RoboDK station: 直线500mm_v50.rdk

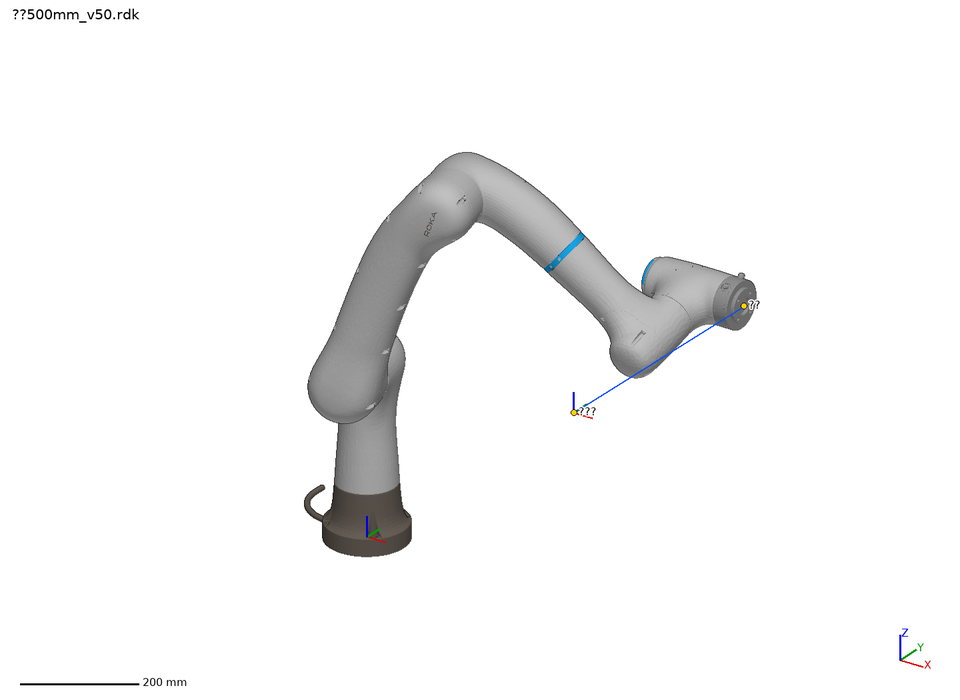
[picture v0: the station drawn from its stored meshes, robots at their saved joint values, targets as dots, program paths as lines]
Station 直线500mm_v50 (saved by RoboDK 5.9.0). Poses are relative to the parent item; angles as X-Y-Z fixed-axis rotations.
  - frame Rokae SR4-C Base at (0, 0, 0) mm
    - robot Rokae SR4-C: 6 axes
        modified DH rows (alpha deg, a mm, theta deg, d mm): 0, 0, 0, 328; -90, 0, -82.875, 0; 0, 400, -97.125, 0; -90, 50, 0, 400; 90, 0, 0, 136; -90, 0, 180, 103.5
        joint limits [-360, -160, -170, -200, -360, -360] to [360, 150, 140, 360, 360, 360]; home [0, 0, -90, 0, 0, 0]; saved at [13.445, 18.79, -111.957, 20.116, 42.538, -15.103]
      - tool , TCP at (0, 0, 0) mm
    - frame 直线运动1坐标系 at (600, -250, 500) mm
      - target 起始点 (Cartesian target) at (0, 0, 0) mm, rotated rx 0 ry 90 rz 0 deg; joints [-32.271, 21.015, -84.736, -66.737, 35.533, 62.153] of Rokae SR4-C
      - target 终点 (Cartesian target) at (0, 500, 0) mm, rotated rx 0 ry 90 rz 0 deg; joints [13.445, 18.79, -111.957, 20.116, 42.538, -15.103] of Rokae SR4-C
  - program 程序1 (5 instructions, listed below)

--- program 程序1 (robot Rokae SR4-C) ---
  设置参考: 直线运动1坐标系
  设置工具 at (0, 0, 0) mm
  MoveJ (起始点)
  设置速度（50.0 mm/s)
  MoveL (终点)
